RoboDK station: Assistive_UR5e_Sergi.rdk

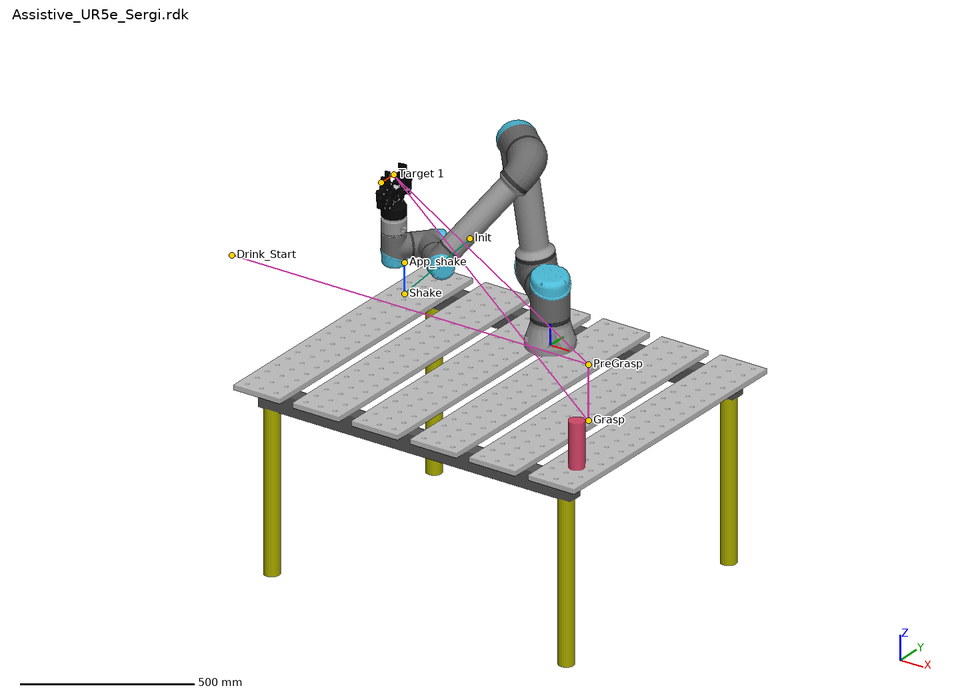
[picture v0: the station drawn from its stored meshes, robots at their saved joint values, targets as dots, program paths as lines]
Station Assistive_UR5e_Sergi (saved by RoboDK 5.9.2). Poses are relative to the parent item; angles as X-Y-Z fixed-axis rotations.
  - frame UR5e Base at (0, 0, 0) mm
    - robot UR5e: 6 axes, payload 5 kg, reach 850 mm, repeatability 0.03 mm, weight 18.4 kg
        modified DH rows (alpha deg, a mm, theta deg, d mm): 0, 0, 0, 162.5; 90, 0, 180, 0; 0, 425, 0, 0; 0, 392.25, 0, 133.3; -90, 0, 0, 99.7; 90, 0, 180, 99.6
        joint limits [-360, -360, -360, -360, -360, -360] to [360, 360, 360, 360, 360, 360]; home [0, -90, -90, 0, 90, 0]; saved at [-130.679, -97.378, -128.12, 315.498, -90, 130.679]
      - tool RobotiQ 2F-85 Gripper (Open), TCP at (0, 0, 130) mm, size 147.4 x 75 x 146.8 mm
      - tool RobotiQ 2F-85 Gripper (Closed), TCP at (0, 0, 130) mm, size 134.4 x 75 x 157.6 mm
    - target Target 1 (Cartesian target) at (-380.86, -238.62, 533.82) mm, rotated rx 0 ry 0 rz 90 deg; joints [-130.679, -89.195, -122.013, 301.208, -90, 130.679] of UR5e
    - target Home (Cartesian target) at (-380.86, -238.62, 533.82) mm, rotated rx 0 ry 0 rz 90 deg; joints [-130.679, -89.195, -122.013, 301.208, -90, 130.679] of UR5e
    - target PreGrasp (Cartesian target) at (511.69, -539.16, 297.03) mm, rotated rx 95.26 ry -4.02 rz 3.58 deg; joints [129.98, -44.106, 83.067, 147.522, -125.856, 187.849] of UR5e
    - target Grasp (Cartesian target) at (511.69, -539.16, 117.03) mm, rotated rx 95.26 ry -4.02 rz 3.58 deg; joints [134.741, -30.853, 91.35, 126.423, -130.585, 188.556] of UR5e
    - target Drink_Start (Cartesian target) at (-738.31, -539.16, 297.03) mm, rotated rx 93.07 ry 5.87 rz -96.08 deg; joints [37.801, -27.14, 49.076, 162.316, -134.115, 177.083] of UR5e
    - target Drink_End (Cartesian target) at (-738.32, -539.16, 297.03) mm, rotated rx 143.07 ry 5.87 rz -96.08 deg; joints [34.28, -36.861, 34.389, 245.485, -116.834, 211.844] of UR5e
  - frame World at (0, 0, 0) mm
    - object Table at (0, 0, 0) mm, size 1193.8 x 965.2 x 609.6 mm, geometry from welding_table.sld
    - target Init (Cartesian target) at (0, -400, 500) mm, rotated rx 90 ry 0 rz 0 deg; joints [-57.836, -65.392, -107.167, 172.559, -57.836, 0] of UR5e
    - target App_shake (joint target) at (-300, -300, 300) mm, rotated rx 90 ry 0 rz 0 deg; joints [-129.97, -84.968, -123.366, -151.667, -129.97, 0] of UR5e
    - target Shake (joint target) at (-300, -300, 200) mm, rotated rx 90 ry 0 rz 0 deg; joints [-129.97, -95.332, -131.473, -133.195, -129.97, 0] of UR5e
    - target App_give5 (joint target) at (-380.86, -238.62, 533.82) mm, rotated rx 0 ry 0 rz 90 deg; joints [-130.679, -89.195, -122.013, 301.208, -90, 130.679] of UR5e
    - target Give5 (joint target) at (-380.86, -300, 533.82) mm, rotated rx 0 ry 0 rz 90 deg; joints [-125.814, -94.091, -116.939, 301.03, -90, 125.814] of UR5e
    - target Target 6 (Cartesian target) at (-380.86, -238.62, 533.82) mm, rotated rx 0 ry 0 rz 90 deg; joints [-130.679, -89.195, -122.013, 301.208, -90, 130.679] of UR5e
  - program Init (3 instructions, listed below)
  - program Hand_shake (5 instructions, listed below)
  - program Give_me_5! (5 instructions, listed below)
  - program MainProgram (4 instructions, listed below)
  - program Pulsar_Boton (4 instructions, listed below)
  - program Bring_Glass (18 instructions, listed below)
  - object Glass at (520, -610, 0) mm, size 50 x 50 x 150 mm, geometry from Cylinder-50x150mm.sld
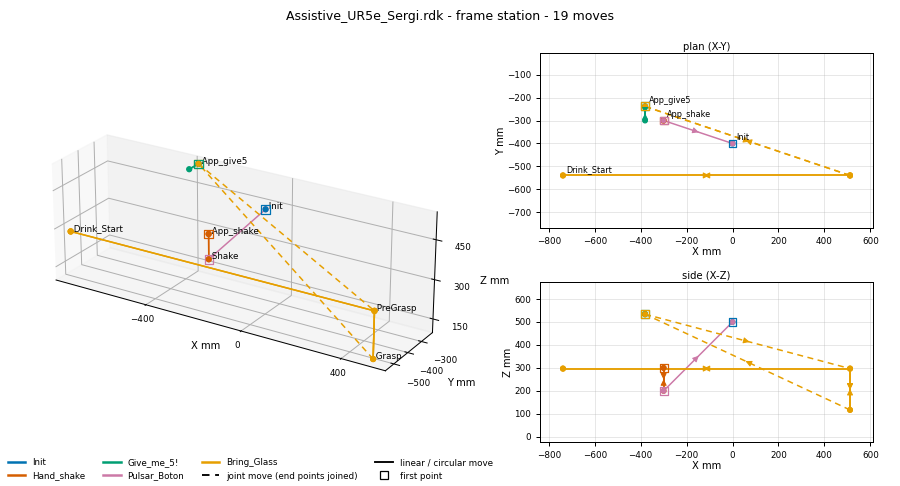
[picture p0: tool path of Assistive_UR5e_Sergi.rdk in frame station, 19 of 19 moves have a stored position in this frame; points joined in program order, loops and branches not executed]

--- program Init (robot UR5e) ---
  Est. Ref.: UR5e Base
  Est. herr: Hand at (0, 0, 50) mm
  MoveJ (Init)

--- program Hand_shake (robot UR5e) ---
  Est. Ref.: UR5e Base
  Est. herr: Hand at (0, 0, 50) mm
  MoveL (App_shake)
  MoveL (Shake)
  MoveL (App_shake)

--- program Give_me_5! (robot UR5e) ---
  Est. Ref.: UR5e Base
  Est. herr: Hand at (0, 0, 50) mm
  MoveL (App_give5)
  MoveL (Give5)
  MoveL (App_give5)

--- program MainProgram (robot UR5e) ---
  Llamar Init
  Llamar Hand_shake
  Llamar Give_me_5!
  Llamar Init

--- program Pulsar_Boton (robot UR5e) ---
  Est. Ref.: UR5e Base
  Est. herr: Hand at (0, 0, 50) mm
  MoveL (Shake)
  MoveL (Init)

--- program Bring_Glass (robot UR5e) ---
  Est. Ref.: UR5e Base
  MoveJ (Home)
  MoveJ (PreGrasp)
  MoveL (Grasp)
  Est. herr: RobotiQ 2F-85 Gripper (Closed)
  Adjuntar a RobotiQ 2F-85 Gripper (Closed)
  MoveL (PreGrasp)
  MoveL (Drink_Start)
  Establecer velocidad (5.0 mm/s)
  MoveL (Drink_End)
  Establecer velocidad (50.0 mm/s)
  Pausa 3.0 s
  MoveL (Drink_Start)
  MoveL (PreGrasp)
  MoveL (Grasp)
  Est. herr: RobotiQ 2F-85 Gripper (Open)
  Separar de RobotiQ 2F-85 Gripper (Closed)
  MoveJ (Home)
